{attribute 'qualified_only'}
VAR_GLOBAL

	bSafetyErrorAck 	AT %Q* : BOOL;
	bAXSafetyErrorAck 	AT %Q* : BOOL;
	bSafetyRun			AT %Q* : BOOL;
	bSafetyRestart		AT %Q* : BOOL;

END_VAR

(* stored: Version 1.1.0.1, ProductVersion 3.1.4024.12
   GVL Safety: Id {7dbc874b-a0ba-482d-92aa-31c8e59bdab6} *)
